% RSLogix 500 project Project_6.RSS, saved by version 8.30.00.16 %
PROJECT "UNTITLED"    % processor: Bul.1763 MicroLogix 1100 Series B %

PROGRAM FILES
  LAD 2   17 rungs

DATA FILES
  O0 OUTPUT  4 elements
  I1 INPUT  6 elements
  S2 STATUS  66 elements
  B3 BINARY  1 elements
  T4 TIMER  1 elements
  C5 COUNTER  1 elements
  R6 CONTROL  1 elements
  N7 INTEGER  4 elements
  F8 FLOAT  1 elements

LADDER 2
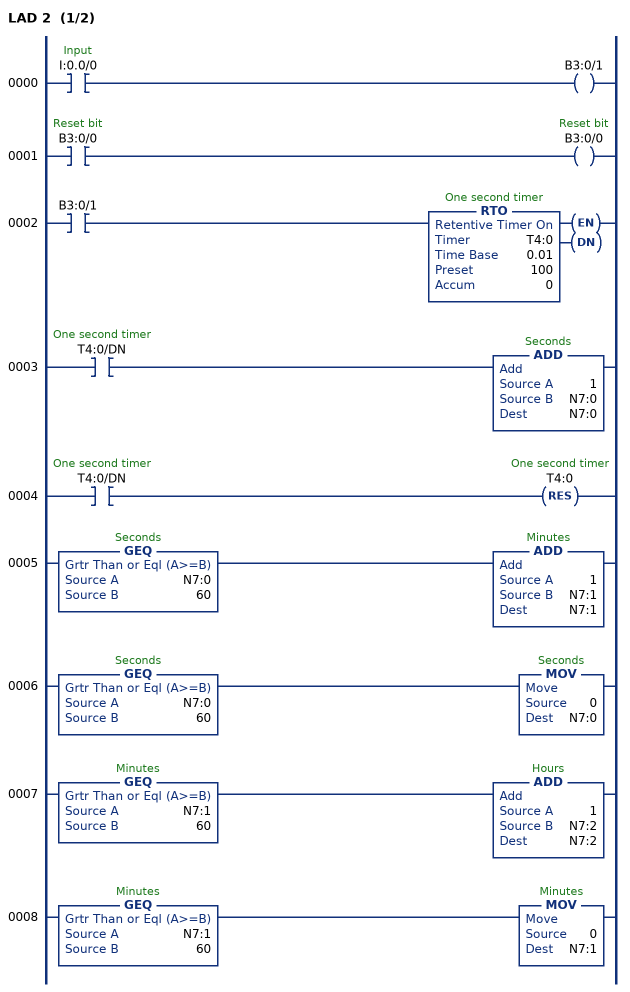
% Rung: 0 %
SOR XIC I:0.0/0 OTE B3:0/1 EOR
%   I:0.0/0  "Input" %
% Rung: 1 %
SOR XIC B3:0/0 OTE B3:0/0 EOR
%   B3:0/0  "Reset bit" %
% Rung: 2 %
SOR XIC B3:0/1 RTO T4:0 0.01 100 0 EOR
%   T4:0  "One second timer" %
% Rung: 3 %
SOR XIC T4:0/DN ADD 1 N7:0 N7:0 EOR
%   T4:0  "One second timer" %
%   N7:0  "Seconds" %
% Rung: 4 %
SOR XIC T4:0/DN RES T4:0 EOR
%   T4:0  "One second timer" %
% Rung: 5 %
SOR GEQ N7:0 60 ADD 1 N7:1 N7:1 EOR
%   N7:0  "Seconds" %
%   N7:1  "Minutes" %
% Rung: 6 %
SOR GEQ N7:0 60 MOV 0 N7:0 EOR
%   N7:0  "Seconds" %
% Rung: 7 %
SOR GEQ N7:1 60 ADD 1 N7:2 N7:2 EOR
%   N7:1  "Minutes" %
%   N7:2  "Hours" %
% Rung: 8 %
SOR GEQ N7:1 60 MOV 0 N7:1 EOR
%   N7:1  "Minutes" %

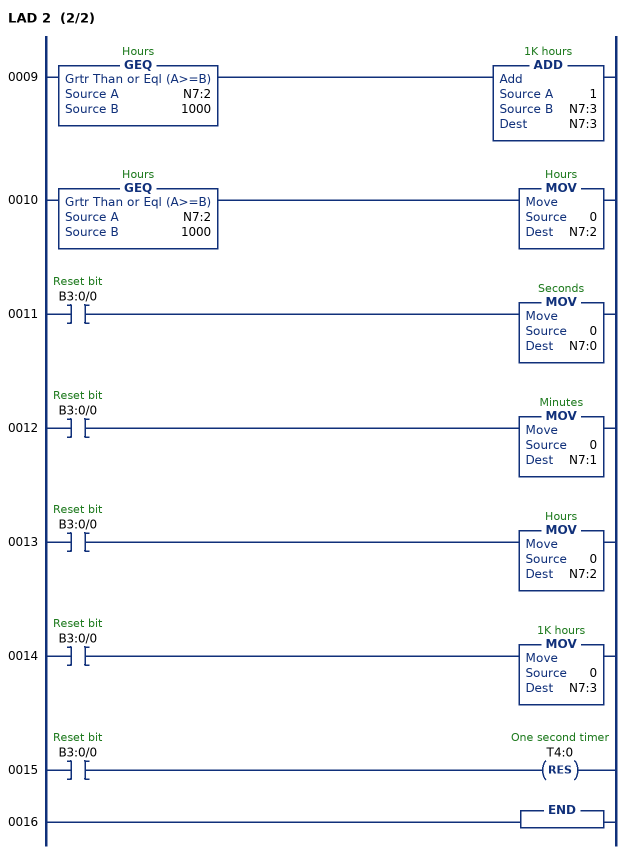
% Rung: 9 %
SOR GEQ N7:2 1000 ADD 1 N7:3 N7:3 EOR
%   N7:2  "Hours" %
%   N7:3  "1K hours" %
% Rung: 10 %
SOR GEQ N7:2 1000 MOV 0 N7:2 EOR
%   N7:2  "Hours" %
% Rung: 11 %
SOR XIC B3:0/0 MOV 0 N7:0 EOR
%   B3:0/0  "Reset bit" %
%   N7:0  "Seconds" %
% Rung: 12 %
SOR XIC B3:0/0 MOV 0 N7:1 EOR
%   B3:0/0  "Reset bit" %
%   N7:1  "Minutes" %
% Rung: 13 %
SOR XIC B3:0/0 MOV 0 N7:2 EOR
%   B3:0/0  "Reset bit" %
%   N7:2  "Hours" %
% Rung: 14 %
SOR XIC B3:0/0 MOV 0 N7:3 EOR
%   B3:0/0  "Reset bit" %
%   N7:3  "1K hours" %
% Rung: 15 %
SOR XIC B3:0/0 RES T4:0 EOR
%   B3:0/0  "Reset bit" %
%   T4:0  "One second timer" %
% Rung: 16 %
SOR END EOR

DATA TABLE (non-zero values as saved)
DATA B3
% B3:0 % 0X0003
DATA T4
% .PRE .ACC %
% T4:0 % 100 0
